Fanuc KAREL source: KA00177.KL

PROGRAM KA00177
%NOLOCKGROUP
VAR
  SRC: ARRAY[4] OF STRING[20]
  DST: ARRAY[4] OF SHORT
BEGIN
  DST = SRC
END KA00177
